(* PLC project Unnamed, Unknown Unnamed 1 *)
(* stored: creationDateTime 2025-03-23T17:08:44, modificationDateTime 2025-04-07T00:54:42 *)

PROGRAM LadderLogic
  VAR
    B_JOG_UP AT %IX1.1 : BOOL;
    B_JOG_DOWN AT %IX1.2 : BOOL;
    B_JOG_CW AT %IX1.3 : BOOL;
    B_JOG_CCW AT %IX1.4 : BOOL;
    B_RESET AT %IX1.5 : BOOL;
    B_START AT %IX1.6 : BOOL;
    MAINT_MODE AT %IX1.7 : BOOL := 1;
    LIM_1 AT %IX2.0 : BOOL;
    LIM_2 AT %IX2.1 : BOOL;
    LIM_3 AT %IX2.2 : BOOL;
    LIM_4 AT %IX2.3 : BOOL;
    ARD_CHECKPOINT AT %IX2.4 : BOOL;
    B_STOP_CYCLE AT %IX2.5 : BOOL;
    B_SOFT_STOP AT %IX2.6 : BOOL;
    B_ESTOP AT %IX2.7 : BOOL := 1;
    LED_MAINT AT %QX1.6 : BOOL;
    LED_AUTO AT %QX1.7 : BOOL;
    LED_ESTOP AT %QX2.0 : BOOL;
    LED_RESET AT %QX2.1 : BOOL;
    LED_POS_DIS AT %QX2.2 : BOOL;
    LED_HOMING AT %QX2.3 : BOOL := 0;
    LED_RUNNING AT %QX2.5 : BOOL := 0;
    PROG_ESTOP AT %QX2.7 : BOOL := 0;
  END_VAR
  VAR
    POWER_ON_FLAG : BOOL;
    BEGIN_HOMING_FLAG : BOOL;
  END_VAR
  VAR_EXTERNAL
    ARD_LIM_1 : BOOL;
    ARD_LIM_2 : BOOL;
  END_VAR
  VAR
    STOP_CYCLE_F : BOOL;
    BLINK_ESTOP : BOOL := 0;
    SOLID_ESTOP : BOOL := 0;
    BLINK_RESET_SLOW : BOOL;
    BLINK_RESET_FAST : BOOL;
    TURN_OFF_RESET_LED : BOOL := 1;
    CAN_RESET : BOOL := 0;
    CAN_HOME : BOOL := 0;
    HOMING_SEQ_1_1 : BOOL := 0;
    HOMING_SEQ_1_2 : BOOL := 0;
  END_VAR
  VAR_EXTERNAL
    ARD_HOMING_2 : BOOL;
  END_VAR
  VAR
    CAN_RESET_SOFT_STOP : BOOL;
    SOLID_HOMING : BOOL;
    BLINK_HOMING : BOOL;
    BLINK_RUNNING : BOOL;
    SOLID_RUNNING : BOOL;
    CAN_AUTO_MOVE : BOOL;
    BEGIN_AUTO_MOVE : BOOL;
  END_VAR
  VAR_EXTERNAL
    ARD_AUTO_MOVING : BOOL;
  END_VAR
  VAR
    CAN_AUTO_UP : BOOL;
  END_VAR
  VAR_EXTERNAL
    ARD_AUTO_UP : BOOL;
  END_VAR
  VAR
    CAN_AUTO_SPIN : BOOL;
  END_VAR
  VAR_EXTERNAL
    ARD_AUTO_SPIN : BOOL;
  END_VAR
  VAR
    CAN_AUTO_DOWN : BOOL;
  END_VAR
  VAR_EXTERNAL
    ARD_AUTO_DOWN : BOOL;
  END_VAR
  VAR
    CAN_AUTO_LOADING : BOOL;
  END_VAR
  VAR_EXTERNAL
    ARD_AUTO_LOADING : BOOL;
    HOMING : BOOL;
    M_MAINT_UP : BOOL;
    M_MAINT_DOWN : BOOL;
    M_MAINT_CW : BOOL;
    M_MAINT_CCW : BOOL;
    ARD_M1_HOME : BOOL;
    ARD_M2_HOME : BOOL;
    ARD_SOFT_STOP : BOOL;
    ARD_ESTOPPED : BOOL;
    ARD_MAINT_MODE : BOOL;
  END_VAR
  VAR
    TON3 : TON;
    TOF3 : TOF;
    TON4 : TON;
    TOF4 : TOF;
    TON0 : TON;
    TON1 : TON;
    TOF5 : TOF;
    TON5 : TON;
    TOF6 : TOF;
    TON6 : TON;
  END_VAR
  VAR  (* added by the conversion: wires and edge detectors of the diagram *)
    _SUB_TIME129_ENO : BOOL;
    _SUB_TIME129_OUT : TIME;
    _SUB_TIME23_ENO : BOOL;
    _SUB_TIME23_OUT : TIME;
    _MAX134_OUT : TIME;
  END_VAR

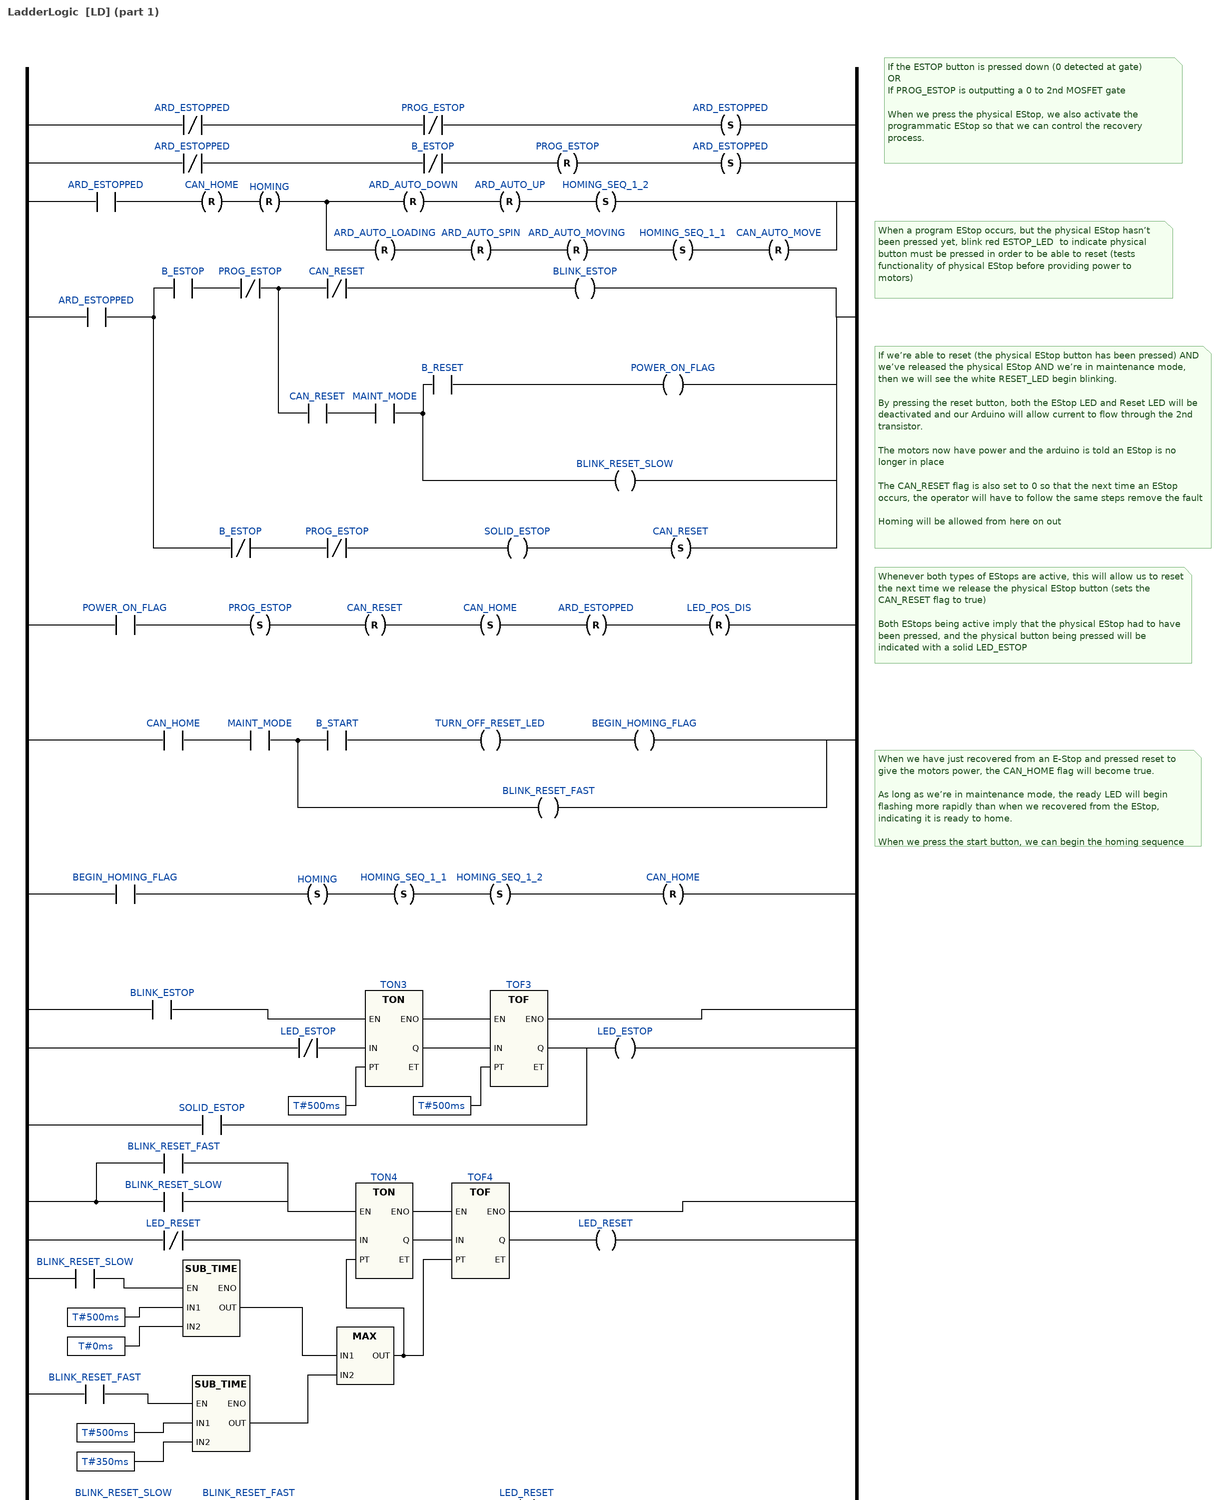
(* LD diagram, written out as Structured Text *)
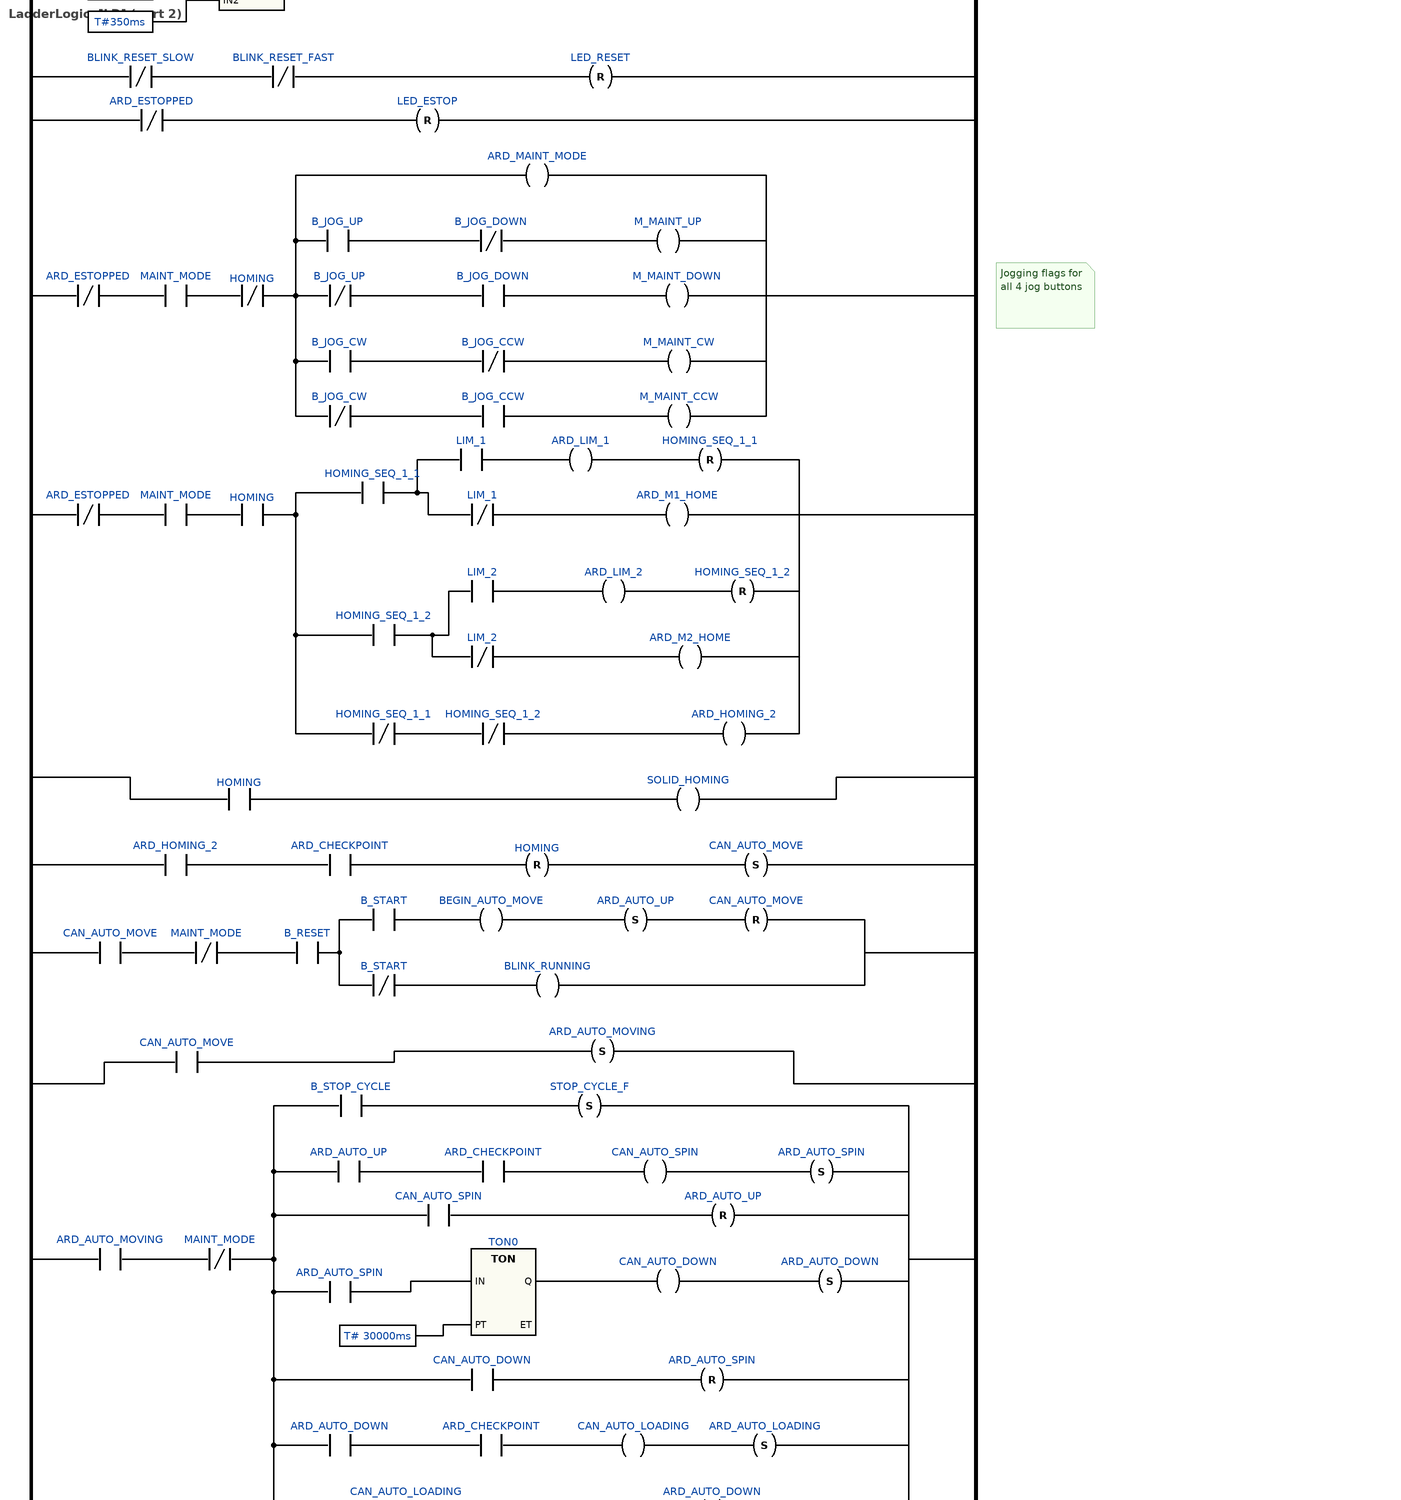
(* If the ESTOP button is pressed down (0 detected at gate)
OR
If PROG_ESTOP is outputting a 0 to 2nd MOSFET gate

When we press the physical EStop, we also activate the programmatic EStop so that we can control the recovery process. *)
(* When a program EStop occurs, but the physical EStop hasn’t been pressed yet, blink red ESTOP_LED  to indicate physical button must be pressed in order to be able to reset (tests functionality of physical EStop before providing power to motors) *)
(* If we’re able to reset (the physical EStop button has been pressed) AND we’ve released the physical EStop AND we’re in maintenance mode, then we will see the white RESET_LED begin blinking.

By pressing the reset button, both the EStop LED and Reset LED will be deactivated and our Arduino will allow current to flow through the 2nd transistor.

The motors now have power and the arduino is told an EStop is no longer in place

The CAN_RESET flag is also set to 0 so that the next time an EStop occurs, the operator will have to follow the same steps remove the fault

Homing will be allowed from here on out *)
(* Whenever both types of EStops are active, this will allow us to reset the next time we release the physical EStop button (sets the CAN_RESET flag to true)

Both EStops being active imply that the physical EStop had to have been pressed, and the physical button being pressed will be indicated with a solid LED_ESTOP *)
(* When we have just recovered from an E-Stop and pressed reset to give the motors power, the CAN_HOME flag will become true.

As long as we’re in maintenance mode, the ready LED will begin flashing more rapidly than when we recovered from the EStop, indicating it is ready to home.

When we press the start button, we can begin the homing sequence *)
(* Jogging flags for all 4 jog buttons *)
M_MAINT_CW := NOT ARD_ESTOPPED AND MAINT_MODE AND NOT HOMING AND B_JOG_CW AND NOT B_JOG_CCW;
M_MAINT_CCW := NOT ARD_ESTOPPED AND MAINT_MODE AND NOT HOMING AND NOT B_JOG_CW AND B_JOG_CCW;
ARD_MAINT_MODE := NOT ARD_ESTOPPED AND MAINT_MODE AND NOT HOMING;
IF NOT ARD_ESTOPPED AND NOT PROG_ESTOP THEN ARD_ESTOPPED := TRUE; END_IF;
M_MAINT_UP := NOT ARD_ESTOPPED AND MAINT_MODE AND NOT HOMING AND B_JOG_UP AND NOT B_JOG_DOWN;
M_MAINT_DOWN := NOT ARD_ESTOPPED AND MAINT_MODE AND NOT HOMING AND NOT B_JOG_UP AND B_JOG_DOWN;
POWER_ON_FLAG := ARD_ESTOPPED AND B_ESTOP AND NOT PROG_ESTOP AND CAN_RESET AND MAINT_MODE AND B_RESET;
IF ARD_ESTOPPED AND NOT B_ESTOP AND NOT PROG_ESTOP THEN CAN_RESET := TRUE; END_IF;
BLINK_RESET_SLOW := ARD_ESTOPPED AND B_ESTOP AND NOT PROG_ESTOP AND CAN_RESET AND MAINT_MODE;
BEGIN_HOMING_FLAG := CAN_HOME AND MAINT_MODE AND B_START;
BLINK_RESET_FAST := CAN_HOME AND MAINT_MODE;
TON3(EN := BLINK_ESTOP, IN := NOT LED_ESTOP, PT := T#500ms);
TOF3(EN := TON3.ENO, IN := TON3.Q, PT := T#500ms);
LED_ESTOP := TOF3.Q OR SOLID_ESTOP;
BLINK_ESTOP := ARD_ESTOPPED AND B_ESTOP AND NOT PROG_ESTOP AND NOT CAN_RESET;
SOLID_ESTOP := ARD_ESTOPPED AND NOT B_ESTOP AND NOT PROG_ESTOP;
_SUB_TIME129_OUT := SUB_TIME(EN := BLINK_RESET_SLOW, IN1 := T#500ms, IN2 := T#0ms, ENO => _SUB_TIME129_ENO);
_SUB_TIME23_OUT := SUB_TIME(EN := BLINK_RESET_FAST, IN1 := T#500ms, IN2 := T#350ms, ENO => _SUB_TIME23_ENO);
_MAX134_OUT := MAX(_SUB_TIME129_OUT, _SUB_TIME23_OUT);
TON4(EN := BLINK_RESET_SLOW OR BLINK_RESET_FAST, IN := NOT LED_RESET, PT := _MAX134_OUT);
TOF4(EN := TON4.ENO, IN := TON4.Q, PT := _MAX134_OUT);
LED_RESET := TOF4.Q;
IF NOT ARD_ESTOPPED AND NOT B_ESTOP THEN PROG_ESTOP := FALSE; END_IF;
IF NOT ARD_ESTOPPED AND NOT B_ESTOP THEN ARD_ESTOPPED := TRUE; END_IF;
IF POWER_ON_FLAG THEN PROG_ESTOP := TRUE; END_IF;
IF POWER_ON_FLAG THEN CAN_RESET := FALSE; END_IF;
IF POWER_ON_FLAG THEN CAN_HOME := TRUE; END_IF;
IF POWER_ON_FLAG THEN ARD_ESTOPPED := FALSE; END_IF;
TURN_OFF_RESET_LED := CAN_HOME AND MAINT_MODE AND B_START;
IF BEGIN_HOMING_FLAG THEN CAN_HOME := FALSE; END_IF;
IF BEGIN_HOMING_FLAG THEN HOMING := TRUE; END_IF;
IF ARD_ESTOPPED THEN CAN_HOME := FALSE; END_IF;
IF ARD_ESTOPPED THEN HOMING := FALSE; END_IF;
IF NOT BLINK_RESET_SLOW AND NOT BLINK_RESET_FAST THEN LED_RESET := FALSE; END_IF;
IF NOT ARD_ESTOPPED THEN LED_ESTOP := FALSE; END_IF;
ARD_LIM_1 := NOT ARD_ESTOPPED AND MAINT_MODE AND HOMING AND HOMING_SEQ_1_1 AND LIM_1;
ARD_LIM_2 := NOT ARD_ESTOPPED AND MAINT_MODE AND HOMING AND HOMING_SEQ_1_2 AND LIM_2;
ARD_M1_HOME := NOT ARD_ESTOPPED AND MAINT_MODE AND HOMING AND HOMING_SEQ_1_1 AND NOT LIM_1;
ARD_M2_HOME := NOT ARD_ESTOPPED AND MAINT_MODE AND HOMING AND HOMING_SEQ_1_2 AND NOT LIM_2;
IF BEGIN_HOMING_FLAG THEN HOMING_SEQ_1_1 := TRUE; END_IF;
IF BEGIN_HOMING_FLAG THEN HOMING_SEQ_1_2 := TRUE; END_IF;
IF NOT ARD_ESTOPPED AND MAINT_MODE AND HOMING AND HOMING_SEQ_1_1 AND LIM_1 THEN HOMING_SEQ_1_1 := FALSE; END_IF;
IF NOT ARD_ESTOPPED AND MAINT_MODE AND HOMING AND HOMING_SEQ_1_2 AND LIM_2 THEN HOMING_SEQ_1_2 := FALSE; END_IF;
ARD_HOMING_2 := NOT ARD_ESTOPPED AND MAINT_MODE AND HOMING AND NOT HOMING_SEQ_1_1 AND NOT HOMING_SEQ_1_2;
SOLID_HOMING := HOMING;
IF ARD_HOMING_2 AND ARD_CHECKPOINT THEN HOMING := FALSE; END_IF;
IF ARD_HOMING_2 AND ARD_CHECKPOINT THEN CAN_AUTO_MOVE := TRUE; END_IF;
IF CAN_AUTO_MOVE AND NOT MAINT_MODE AND B_RESET AND B_START THEN ARD_AUTO_UP := TRUE; END_IF;
IF CAN_AUTO_MOVE AND NOT MAINT_MODE AND B_RESET AND B_START THEN CAN_AUTO_MOVE := FALSE; END_IF;
IF ARD_AUTO_MOVING AND NOT MAINT_MODE AND ARD_AUTO_UP AND ARD_CHECKPOINT THEN ARD_AUTO_SPIN := TRUE; END_IF;
TON0(IN := ARD_AUTO_MOVING AND NOT MAINT_MODE AND ARD_AUTO_SPIN, PT := T# 30000ms);
CAN_AUTO_DOWN := TON0.Q;
IF TON0.Q THEN ARD_AUTO_DOWN := TRUE; END_IF;
CAN_AUTO_LOADING := ARD_AUTO_MOVING AND NOT MAINT_MODE AND ARD_AUTO_DOWN AND ARD_CHECKPOINT;
IF ARD_AUTO_MOVING AND NOT MAINT_MODE AND ARD_AUTO_DOWN AND ARD_CHECKPOINT THEN ARD_AUTO_LOADING := TRUE; END_IF;
IF ARD_ESTOPPED THEN HOMING_SEQ_1_1 := TRUE; END_IF;
IF ARD_ESTOPPED THEN HOMING_SEQ_1_2 := TRUE; END_IF;
IF ARD_ESTOPPED THEN CAN_AUTO_MOVE := FALSE; END_IF;
IF ARD_ESTOPPED THEN ARD_AUTO_UP := FALSE; END_IF;
IF ARD_ESTOPPED THEN ARD_AUTO_MOVING := FALSE; END_IF;
IF ARD_ESTOPPED THEN ARD_AUTO_DOWN := FALSE; END_IF;
IF ARD_ESTOPPED THEN ARD_AUTO_LOADING := FALSE; END_IF;
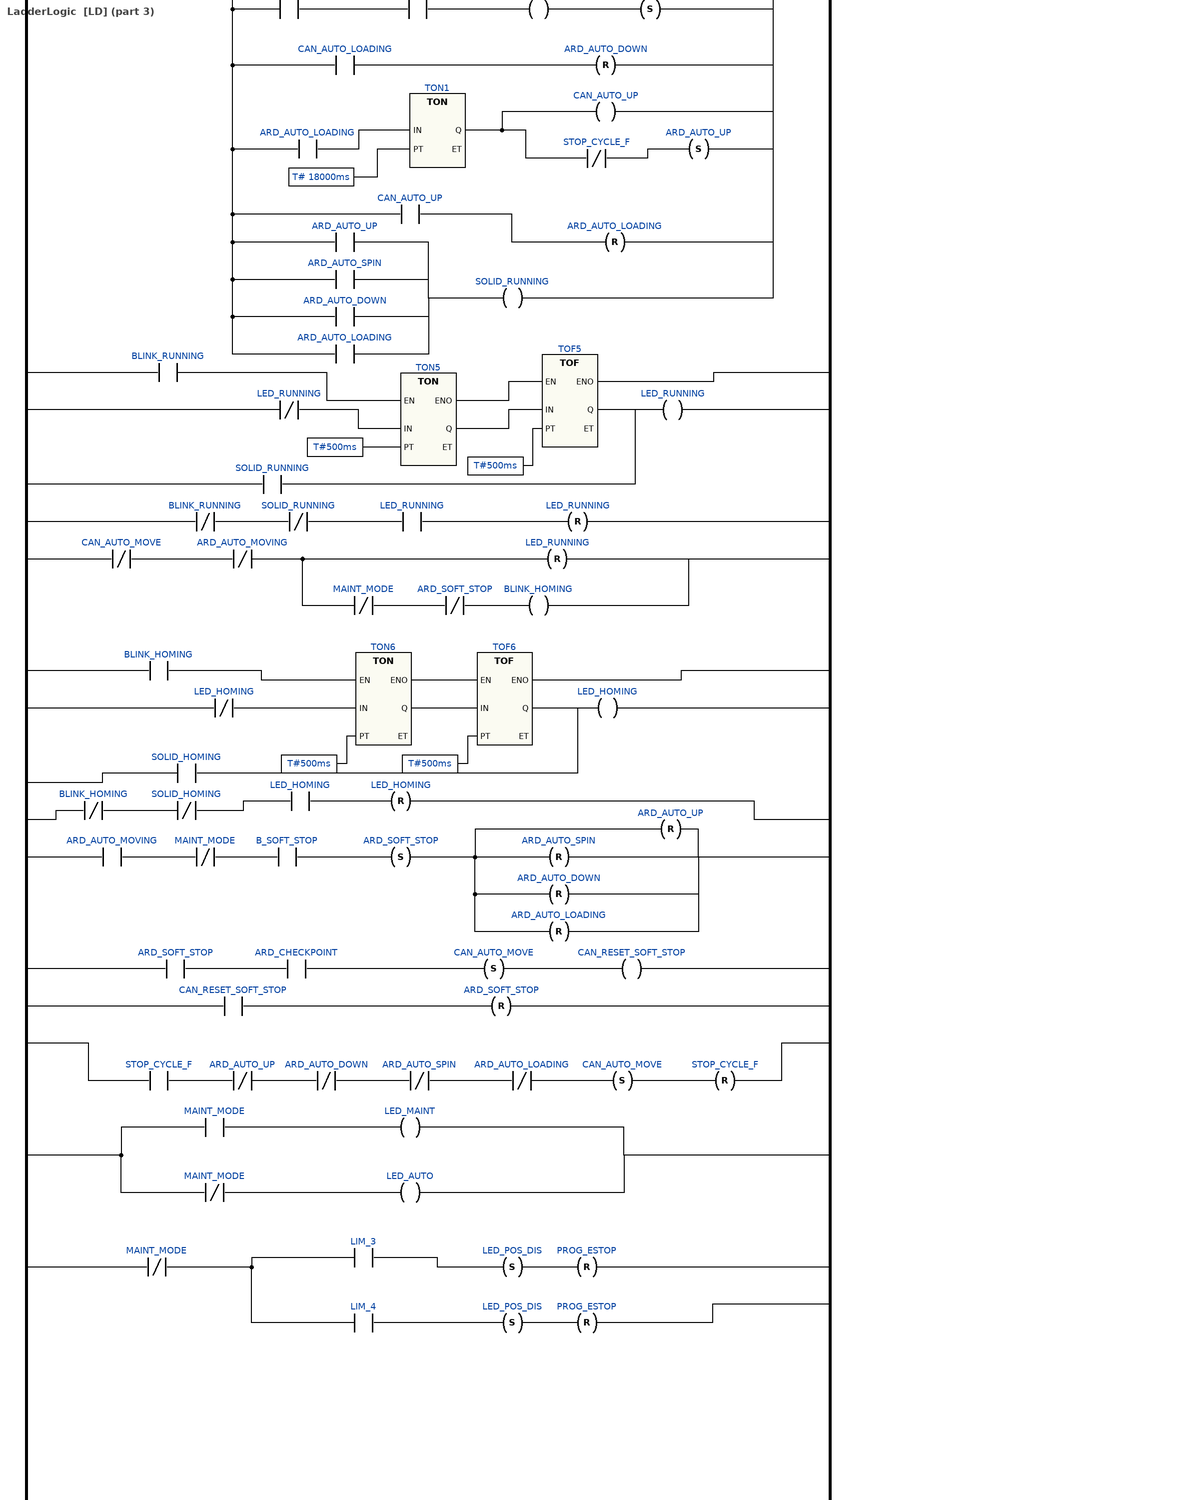
SOLID_RUNNING := ARD_AUTO_MOVING AND NOT MAINT_MODE AND (ARD_AUTO_DOWN OR ARD_AUTO_LOADING OR ARD_AUTO_SPIN OR ARD_AUTO_UP);
IF CAN_AUTO_MOVE THEN ARD_AUTO_MOVING := TRUE; END_IF;
BEGIN_AUTO_MOVE := CAN_AUTO_MOVE AND NOT MAINT_MODE AND B_RESET AND B_START;
IF ARD_AUTO_MOVING AND NOT MAINT_MODE AND CAN_AUTO_SPIN THEN ARD_AUTO_UP := FALSE; END_IF;
CAN_AUTO_SPIN := ARD_AUTO_MOVING AND NOT MAINT_MODE AND ARD_AUTO_UP AND ARD_CHECKPOINT;
IF ARD_AUTO_MOVING AND NOT MAINT_MODE AND CAN_AUTO_DOWN THEN ARD_AUTO_SPIN := FALSE; END_IF;
IF ARD_AUTO_MOVING AND NOT MAINT_MODE AND CAN_AUTO_LOADING THEN ARD_AUTO_DOWN := FALSE; END_IF;
TON1(IN := ARD_AUTO_MOVING AND NOT MAINT_MODE AND ARD_AUTO_LOADING, PT := T# 18000ms);
CAN_AUTO_UP := TON1.Q;
IF ARD_AUTO_MOVING AND NOT MAINT_MODE AND CAN_AUTO_UP THEN ARD_AUTO_LOADING := FALSE; END_IF;
IF ARD_ESTOPPED THEN ARD_AUTO_SPIN := FALSE; END_IF;
BLINK_RUNNING := CAN_AUTO_MOVE AND NOT MAINT_MODE AND B_RESET AND NOT B_START;
TON5(EN := BLINK_RUNNING, IN := NOT LED_RUNNING, PT := T#500ms);
TOF5(EN := TON5.ENO, IN := TON5.Q, PT := T#500ms);
LED_RUNNING := TOF5.Q OR SOLID_RUNNING;
IF NOT CAN_AUTO_MOVE AND NOT ARD_AUTO_MOVING THEN LED_RUNNING := FALSE; END_IF;
BLINK_HOMING := NOT CAN_AUTO_MOVE AND NOT ARD_AUTO_MOVING AND NOT MAINT_MODE AND NOT ARD_SOFT_STOP;
TON6(EN := BLINK_HOMING, IN := NOT LED_HOMING, PT := T#500ms);
TOF6(EN := TON6.ENO, IN := TON6.Q, PT := T#500ms);
LED_HOMING := TOF6.Q OR SOLID_HOMING;
IF ARD_AUTO_MOVING AND NOT MAINT_MODE AND B_SOFT_STOP THEN ARD_SOFT_STOP := TRUE; END_IF;
IF ARD_AUTO_MOVING AND NOT MAINT_MODE AND B_SOFT_STOP THEN ARD_AUTO_UP := FALSE; END_IF;
IF ARD_AUTO_MOVING AND NOT MAINT_MODE AND B_SOFT_STOP THEN ARD_AUTO_SPIN := FALSE; END_IF;
IF ARD_AUTO_MOVING AND NOT MAINT_MODE AND B_SOFT_STOP THEN ARD_AUTO_DOWN := FALSE; END_IF;
IF ARD_AUTO_MOVING AND NOT MAINT_MODE AND B_SOFT_STOP THEN ARD_AUTO_LOADING := FALSE; END_IF;
IF ARD_SOFT_STOP AND ARD_CHECKPOINT THEN CAN_AUTO_MOVE := TRUE; END_IF;
IF CAN_RESET_SOFT_STOP THEN ARD_SOFT_STOP := FALSE; END_IF;
CAN_RESET_SOFT_STOP := ARD_SOFT_STOP AND ARD_CHECKPOINT;
IF NOT BLINK_HOMING AND NOT SOLID_HOMING AND LED_HOMING THEN LED_HOMING := FALSE; END_IF;
IF NOT BLINK_RUNNING AND NOT SOLID_RUNNING AND LED_RUNNING THEN LED_RUNNING := FALSE; END_IF;
IF ARD_AUTO_MOVING AND NOT MAINT_MODE AND B_STOP_CYCLE THEN STOP_CYCLE_F := TRUE; END_IF;
IF TON1.Q AND NOT STOP_CYCLE_F THEN ARD_AUTO_UP := TRUE; END_IF;
IF STOP_CYCLE_F AND NOT ARD_AUTO_UP AND NOT ARD_AUTO_DOWN AND NOT ARD_AUTO_SPIN AND NOT ARD_AUTO_LOADING THEN CAN_AUTO_MOVE := TRUE; END_IF;
IF STOP_CYCLE_F AND NOT ARD_AUTO_UP AND NOT ARD_AUTO_DOWN AND NOT ARD_AUTO_SPIN AND NOT ARD_AUTO_LOADING THEN STOP_CYCLE_F := FALSE; END_IF;
LED_MAINT := MAINT_MODE;
LED_AUTO := NOT MAINT_MODE;
IF NOT MAINT_MODE AND LIM_3 THEN PROG_ESTOP := FALSE; END_IF;
IF NOT MAINT_MODE AND LIM_3 THEN LED_POS_DIS := TRUE; END_IF;
IF POWER_ON_FLAG THEN LED_POS_DIS := FALSE; END_IF;
IF NOT MAINT_MODE AND LIM_4 THEN LED_POS_DIS := TRUE; END_IF;
IF NOT MAINT_MODE AND LIM_4 THEN PROG_ESTOP := FALSE; END_IF;
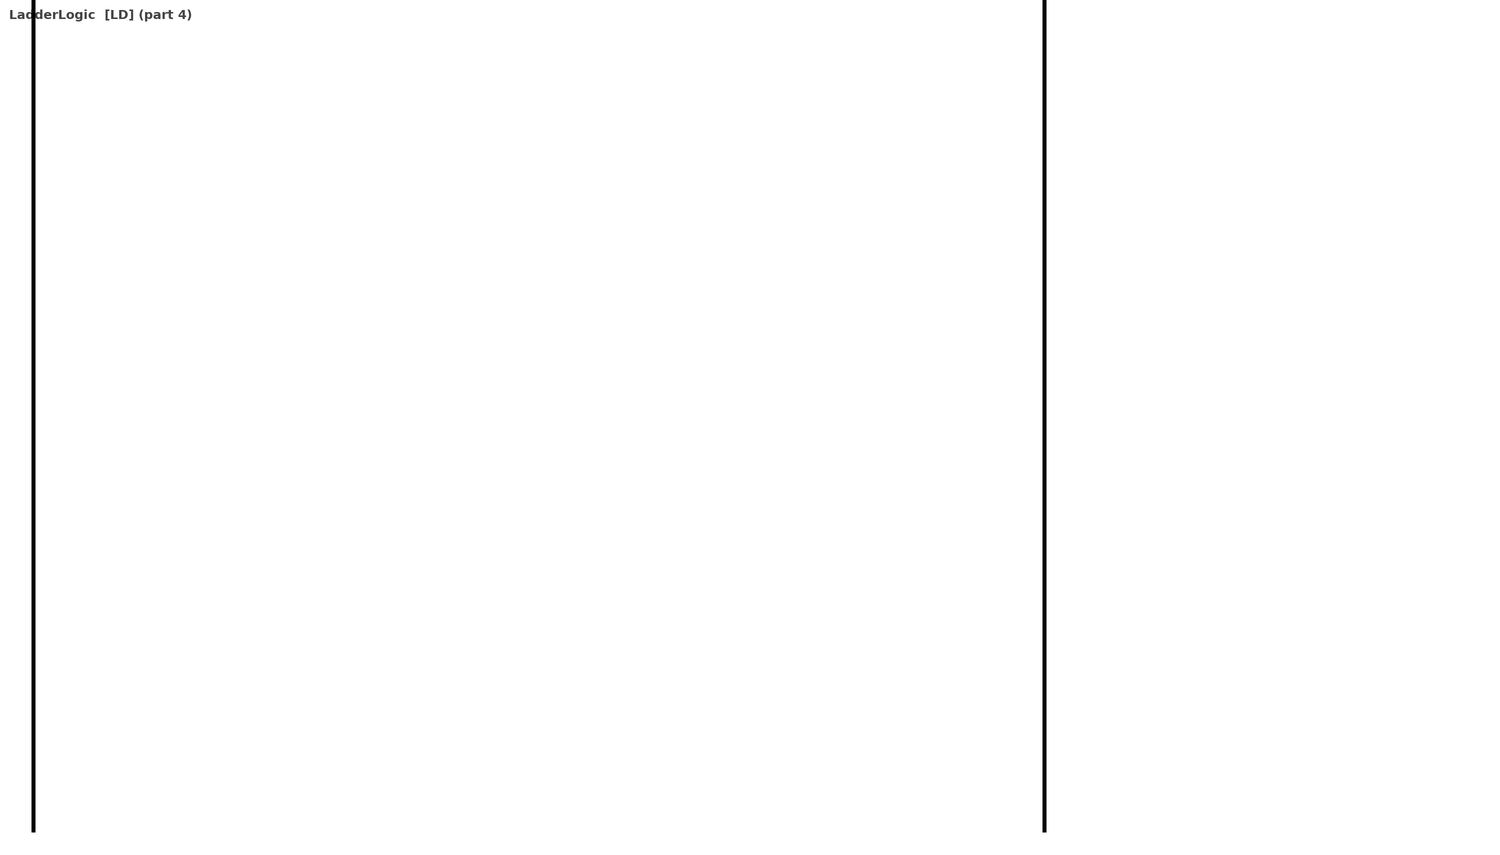
END_PROGRAM

CONFIGURATION Config0
  RESOURCE Res0 ON PLC
    TASK task0(INTERVAL := T#20ms, PRIORITY := 0);
    PROGRAM instance0 WITH task0 : LadderLogic;
  END_RESOURCE
END_CONFIGURATION
